DATA_BLOCK "NG_DB"
{ S7_Optimized_Access := 'TRUE' }
VERSION : 0.1
NON_RETAIN
"NG"

BEGIN

END_DATA_BLOCK

